PROGRAM Read
VAR
	Read_R1				:FB_Lesen;
	Read_R2				:FB_Lesen;
	Read_R3				:FB_Lesen;
	Read_R4				:FB_Lesen;
	Read_R5				:FB_Lesen;
	Read_R6				:FB_Lesen;
	Read_R7				:FB_Lesen;
END_VAR

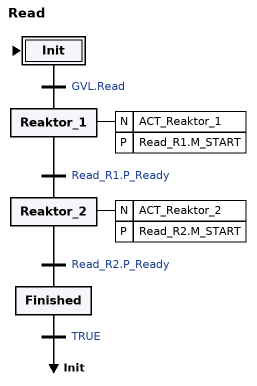
INITIAL_STEP Init:
END_STEP
TRANSITION FROM Init TO Reaktor_1
    := GVL.Read;
END_TRANSITION
STEP Reaktor_1:
    ACT_Reaktor_1(N);
    Read_R1.M_START(P);
END_STEP
TRANSITION FROM Reaktor_1 TO Reaktor_2
    := Read_R1.P_Ready;
END_TRANSITION
STEP Reaktor_2:
    ACT_Reaktor_2(N);
    Read_R2.M_START(P);
END_STEP
TRANSITION FROM Reaktor_2 TO Finished
    := Read_R2.P_Ready;
END_TRANSITION
STEP Finished:
END_STEP
TRANSITION FROM Finished TO Init
    := TRUE;
END_TRANSITION

ACTION ACT_Reaktor_1:
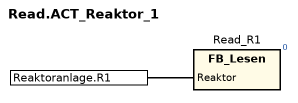
Read_R1(Reaktor := Reaktoranlage.R1); // FB_Lesen
END_ACTION

ACTION ACT_Reaktor_2:
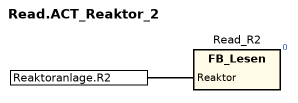
Read_R2(Reaktor := Reaktoranlage.R2); // FB_Lesen
END_ACTION

END_PROGRAM

(* stored: Version 1.1.0.1, ProductVersion 3.1.4024.12
   POU Read: Id {6e8361ab-729c-4f56-af5a-95a9d6e7aa2f}, SpecialFunc None
   Action ACT_Reaktor_1: Id {db11f980-ecfe-45a6-a6be-121808708e90}
   Action ACT_Reaktor_2: Id {5d666480-ad17-48a7-b5da-fb56e7f0f069} *)
